FUNCTION F_VerboseLogger : BOOL
VAR_INPUT
	Message : STRING;
END_VAR

ADSLOGSTR( msgCtrlMask := ADSLOG_MSGTYPE_LOG, msgFmtStr := 'Verbose Msg. : %s', strArg := Message);

END_FUNCTION

(* stored: Version 1.1.0.1, ProductVersion 3.1.4024.12
   POU F_VerboseLogger: Id {cce0ef73-8c43-40aa-8ec6-b58911df9109}, SpecialFunc None *)
